LIN {X 0,Y 71.23,Z 524.249,A -85,B 0,C 180,E1 -30254.281,E2 -30254.281} C_VEL
LIN {X 0,Y 69.533,Z 525.783,A -85,B 0,C 180,E1 -30256.224,E2 -30256.224} C_VEL
LIN {X 0,Y 68.086,Z 526.954,A -85,B 0,C 180,E1 -30257.295,E2 -30257.295} C_VEL
LIN {X 0,Y 57.032,Z 533.486,A -85,B 0,C 180,E1 -30262.453,E2 -30262.453} C_VEL
LIN {X 0,Y 47.989,Z 537.812,A -85,B 0,C 180,E1 -30268.517,E2 -30268.517} C_VEL
LIN {X 0,Y 42.388,Z 540.184,A -85,B 0,C 180,E1 -30274.005,E2 -30274.005} C_VEL
LIN {X 0,Y 37.239,Z 541.987,A -85,B 0,C 180,E1 -30280.983,E2 -30280.983} C_VEL
LIN {X 0,Y 29.54,Z 544.455,A -85,B 0,C 180,E1 -30301.587,E2 -30301.587} C_VEL
LIN {X 0,Y 27.549,Z 545.056,A -85,B 0,C 180,E1 -30315.22,E2 -30315.22} C_VEL
LIN {X 0,Y 27.127,Z 545.222,A -85,B 0,C 180,E1 -30330,E2 -30330} C_VEL
LIN {X 0,Y 27.542,Z 545.056,A -85,B 0,C 180,E1 -30344.783,E2 -30344.783} C_VEL
LIN {X 0,Y 29.537,Z 544.455,A -85,B 0,C 180,E1 -30358.416,E2 -30358.416} C_VEL
LIN {X 0,Y 37.239,Z 541.987,A -85,B 0,C 180,E1 -30379.016,E2 -30379.016} C_VEL
LIN {X 0,Y 45.149,Z 539.032,A -85,B 0,C 180,E1 -30388.885,E2 -30388.885} C_VEL
LIN {X 0,Y 53.969,Z 535.041,A -85,B 0,C 180,E1 -30395.72,E2 -30395.72} C_VEL
LIN {X 0,Y 63.264,Z 529.907,A -85,B 0,C 180,E1 -30400.768,E2 -30400.768} C_VEL
LIN {X 0,Y 68.069,Z 526.953,A -85,B 0,C 180,E1 -30402.751,E2 -30402.751} C_VEL
LIN {X 0,Y 69.534,Z 525.783,A -85,B 0,C 180,E1 -30403.774,E2 -30403.774} C_VEL
LIN {X 0,Y 71.209,Z 524.264,A -85,B 0,C 180,E1 -30405.715,E2 -30405.715} C_VEL
LIN {X 0,Y 72.238,Z 522.956,A -85,B 0,C 180,E1 -30408.777,E2 -30408.777} C_VEL
LIN {X 0,Y 73.193,Z 521.436,A -85,B 0,C 180,E1 -30414.487,E2 -30414.487} C_VEL
LIN {X 0,Y 74.016,Z 520.373,A -85,B 0,C 180,E1 -30419.997,E2 -30419.997} C_VEL
LIN {X 0,Y 72.973,Z 521.245,A -85,B 0,C 180,E1 -30426.486,E2 -30426.486} C_VEL
LIN {X 0,Y 72.133,Z 522.493,A -85,B 0,C 180,E1 -30433.02,E2 -30433.02} C_VEL
LIN {X 0,Y 71.688,Z 523.511,A -85,B 0,C 180,E1 -30437.101,E2 -30437.101} C_VEL
LIN {X 0,Y 70.173,Z 526.051,A -85,B 0,C 180,E1 -30443.613,E2 -30443.613} C_VEL
LIN {X 0,Y 69.168,Z 527.484,A -85,B 0,C 180,E1 -30447.202,E2 -30447.202} C_VEL
LIN {X 0,Y 67.175,Z 530.211,A -85,B 0,C 180,E1 -30453.18,E2 -30453.18} C_VEL
LIN {X 0,Y 63.118,Z 534.913,A -85,B 0,C 180,E1 -30464.295,E2 -30464.295} C_VEL
LIN {X 0,Y 61.528,Z 538.124,A -85,B 0,C 180,E1 -30475.172,E2 -30475.172} C_VEL
LIN {X 0,Y 62.218,Z 540.119,A -85,B 0,C 180,E1 -30484.636,E2 -30484.636} C_VEL
LIN {X 0,Y 66.705,Z 541.924,A -85,B 0,C 180,E1 -30497.836,E2 -30497.836} C_VEL
LIN {X 0,Y 70.834,Z 542.361,A -85,B 0,C 180,E1 -30504.306,E2 -30504.306} C_VEL
LIN {X 0,Y 76.029,Z 542.359,A -85,B 0,C 180,E1 -30510,E2 -30510} C_VEL
LIN {X 0,Y 70.662,Z 542.338,A -85,B 0,C 180,E1 -30515.991,E2 -30515.991} C_VEL
LIN {X 0,Y 65.424,Z 541.656,A -85,B 0,C 180,E1 -30524.819,E2 -30524.819} C_VEL
LIN {X 0,Y 61.967,Z 539.777,A -85,B 0,C 180,E1 -30536.978,E2 -30536.978} C_VEL
LIN {X 0,Y 61.667,Z 537.523,A -85,B 0,C 180,E1 -30547.089,E2 -30547.089} C_VEL
LIN {X 0,Y 64.093,Z 533.66,A -85,B 0,C 180,E1 -30558.864,E2 -30558.864} C_VEL
LIN {X 0,Y 67.132,Z 530.214,A -85,B 0,C 180,E1 -30566.877,E2 -30566.877} C_VEL
LIN {X 0,Y 69.117,Z 527.515,A -85,B 0,C 180,E1 -30572.776,E2 -30572.776} C_VEL
LIN {X 0,Y 70.159,Z 526.06,A -85,B 0,C 180,E1 -30576.382,E2 -30576.382} C_VEL
LIN {X 0,Y 71.673,Z 523.521,A -85,B 0,C 180,E1 -30582.896,E2 -30582.896} C_VEL
LIN {X 0,Y 72.372,Z 522.086,A -85,B 0,C 180,E1 -30588.804,E2 -30588.804} C_VEL
LIN {X 0,Y 73.157,Z 521.071,A -85,B 0,C 180,E1 -30594.49,E2 -30594.49} C_VEL
LIN {X 0,Y 73.978,Z 520.403,A -85,B 0,C 180,E1 -30600.003,E2 -30600.003} C_VEL
LIN {X 0,Y 72.983,Z 521.692,A -85,B 0,C 180,E1 -30606.47,E2 -30606.47} C_VEL
LIN {X 0,Y 71.817,Z 522.781,A -85,B 0,C 180,E1 -30608.611,E2 -30608.611} C_VEL
LIN {X 0,Y 69.339,Z 524.72,A -85,B 0,C 180,E1 -30610.507,E2 -30610.507} C_VEL
LIN {X 0,Y 66.81,Z 526.482,A -85,B 0,C 180,E1 -30611.609,E2 -30611.609} C_VEL
LIN {X 0,Y 56.852,Z 532.194,A -85,B 0,C 180,E1 -30614.584,E2 -30614.584} C_VEL
LIN {X 0,Y 48.207,Z 536.373,A -85,B 0,C 180,E1 -30618.631,E2 -30618.631} C_VEL
LIN {X 0,Y 38.852,Z 539.986,A -85,B 0,C 180,E1 -30625.252,E2 -30625.252} C_VEL
LIN {X 0,Y 33.001,Z 541.789,A -85,B 0,C 180,E1 -30631.589,E2 -30631.589} C_VEL
LIN {X 0,Y 23.518,Z 544.257,A -85,B 0,C 180,E1 -30653.298,E2 -30653.298} C_VEL
LIN {X 0,Y 20.755,Z 544.859,A -85,B 0,C 180,E1 -30670.208,E2 -30670.208} C_VEL
LIN {X 0,Y 20.02,Z 545.025,A -85,B 0,C 180,E1 -30690,E2 -30690} C_VEL
LIN {X 0,Y 20.75,Z 544.859,A -85,B 0,C 180,E1 -30709.797,E2 -30709.797} C_VEL
LIN {X 0,Y 23.516,Z 544.257,A -85,B 0,C 180,E1 -30726.706,E2 -30726.706} C_VEL
LIN {X 0,Y 33.002,Z 541.789,A -85,B 0,C 180,E1 -30748.41,E2 -30748.41} C_VEL
LIN {X 0,Y 41.912,Z 538.834,A -85,B 0,C 180,E1 -30757.255,E2 -30757.255} C_VEL
LIN {X 0,Y 51.452,Z 534.843,A -85,B 0,C 180,E1 -30762.968,E2 -30762.968} C_VEL
LIN {X 0,Y 61.285,Z 529.709,A -85,B 0,C 180,E1 -30767.08,E2 -30767.08} C_VEL
LIN {X 0,Y 64.629,Z 527.791,A -85,B 0,C 180,E1 -30768.146,E2 -30768.146} C_VEL
LIN {X 0,Y 66.463,Z 526.233,A -85,B 0,C 180,E1 -30771.212,E2 -30771.212} C_VEL
LIN {X 0,Y 67.993,Z 524.44,A -85,B 0,C 180,E1 -30779.997,E2 -30779.997} C_VEL
LIN {X 0,Y 67.02,Z 525.123,A -85,B 0,C 180,E1 -30786.016,E2 -30786.016} C_VEL
LIN {X 0,Y 66.141,Z 526.239,A -85,B 0,C 180,E1 -30792.266,E2 -30792.266} C_VEL
LIN {X 0,Y 65.681,Z 526.931,A -85,B 0,C 180,E1 -30795.636,E2 -30795.636} C_VEL
LIN {X 0,Y 63.819,Z 529.051,A -85,B 0,C 180,E1 -30802.408,E2 -30802.408} C_VEL
LIN {X 0,Y 62.355,Z 530.751,A -85,B 0,C 180,E1 -30806.793,E2 -30806.793} C_VEL
LIN {X 0,Y 60.941,Z 532.143,A -85,B 0,C 180,E1 -30810.65,E2 -30810.65} C_VEL
LIN {X 0,Y 56.616,Z 536.128,A -85,B 0,C 180,E1 -30821.859,E2 -30821.859} C_VEL
LIN {X 0,Y 54.917,Z 538.355,A -85,B 0,C 180,E1 -30830.219,E2 -30830.219} C_VEL
LIN {X 0,Y 54.954,Z 540.749,A -85,B 0,C 180,E1 -30843.527,E2 -30843.527} C_VEL
LIN {X 0,Y 58.247,Z 542.165,A -85,B 0,C 180,E1 -30856.036,E2 -30856.036} C_VEL
LIN {X 0,Y 63.437,Z 542.703,A -85,B 0,C 180,E1 -30865.57,E2 -30865.57} C_VEL
LIN {X 0,Y 66.992,Z 542.61,A -85,B 0,C 180,E1 -30870,E2 -30870} C_VEL
LIN {X 0,Y 62.054,Z 542.606,A -85,B 0,C 180,E1 -30876.503,E2 -30876.503} C_VEL
LIN {X 0,Y 58.047,Z 542.141,A -85,B 0,C 180,E1 -30884.414,E2 -30884.414} C_VEL
LIN {X 0,Y 54.953,Z 540.75,A -85,B 0,C 180,E1 -30896.47,E2 -30896.47} C_VEL
LIN {X 0,Y 54.969,Z 538.321,A -85,B 0,C 180,E1 -30909.911,E2 -30909.911} C_VEL
LIN {X 0,Y 59.439,Z 533.499,A -85,B 0,C 180,E1 -30925.858,E2 -30925.858} C_VEL
LIN {X 0,Y 60.902,Z 532.155,A -85,B 0,C 180,E1 -30929.364,E2 -30929.364} C_VEL
LIN {X 0,Y 62.581,Z 530.469,A -85,B 0,C 180,E1 -30933.949,E2 -30933.949} C_VEL
LIN {X 0,Y 63.818,Z 529.043,A -85,B 0,C 180,E1 -30937.636,E2 -30937.636} C_VEL
LIN {X 0,Y 65.679,Z 526.932,A -85,B 0,C 180,E1 -30944.37,E2 -30944.37} C_VEL
LIN {X 0,Y 66.136,Z 526.243,A -85,B 0,C 180,E1 -30947.733,E2 -30947.733} C_VEL
LIN {X 0,Y 67.018,Z 525.125,A -85,B 0,C 180,E1 -30953.984,E2 -30953.984} C_VEL
LIN {X 0,Y 67.974,Z 524.453,A -85,B 0,C 180,E1 -30960.003,E2 -30960.003} C_VEL
LIN {X 0,Y 66.934,Z 525.57,A -85,B 0,C 180,E1 -30966.03,E2 -30966.03} C_VEL
LIN {X 0,Y 66.443,Z 526.249,A -85,B 0,C 180,E1 -30968.811,E2 -30968.811} C_VEL
LIN {X 0,Y 64.638,Z 527.792,A -85,B 0,C 180,E1 -30971.894,E2 -30971.894} C_VEL
LIN {X 0,Y 56.852,Z 532.194,A -85,B 0,C 180,E1 -30974.584,E2 -30974.584} C_VEL
LIN {X 0,Y 51.655,Z 534.66,A -85,B 0,C 180,E1 -30976.114,E2 -30976.114} C_VEL
LIN {X 0,Y 46.14,Z 536.86,A -85,B 0,C 180,E1 -30976.82,E2 -30976.82} C_VEL
LIN {X 0,Y 34.766,Z 540.354,A -85,B 0,C 180,E1 -30978.039,E2 -30978.039} C_VEL
LIN {X 0,Y 28.325,Z 542.039,A -85,B 0,C 180,E1 -30981.502,E2 -30981.502} C_VEL
LIN {X 0,Y 27.465,Z 542.133,A -85,B 0,C 180,E1 -30982.411,E2 -30982.411} C_VEL
LIN {X 0,Y 18.313,Z 544.06,A -85,B 0,C 180,E1 -30999.867,E2 -30999.867} C_VEL
LIN {X 0,Y 14.258,Z 544.661,A -85,B 0,C 180,E1 -31020.468,E2 -31020.468} C_VEL
LIN {X 0,Y 12.927,Z 544.828,A -85,B 0,C 180,E1 -31050,E2 -31050} C_VEL
LIN {X 0,Y 14.254,Z 544.661,A -85,B 0,C 180,E1 -31079.54,E2 -31079.54} C_VEL
LIN {X 0,Y 18.311,Z 544.059,A -85,B 0,C 180,E1 -31100.138,E2 -31100.138} C_VEL
LIN {X 0,Y 29.89,Z 541.591,A -85,B 0,C 180,E1 -31120.134,E2 -31120.134} C_VEL
LIN {X 0,Y 39.705,Z 538.636,A -85,B 0,C 180,E1 -31126.782,E2 -31126.782} C_VEL
LIN {X 0,Y 49.829,Z 534.645,A -85,B 0,C 180,E1 -31130.849,E2 -31130.849} C_VEL
LIN {X 0,Y 58.983,Z 530.129,A -85,B 0,C 180,E1 -31133.466,E2 -31133.466} C_VEL
LIN {X 0,Y 60.842,Z 528.987,A -85,B 0,C 180,E1 -31135.177,E2 -31135.177} C_VEL
LIN {X 0,Y 61.729,Z 528.247,A -85,B 0,C 180,E1 -31139.996,E2 -31139.996} C_VEL
LIN {X 0,Y 60.611,Z 528.88,A -85,B 0,C 180,E1 -31146.655,E2 -31146.655} C_VEL
LIN {X 0,Y 59.556,Z 529.947,A -85,B 0,C 180,E1 -31153.648,E2 -31153.648} C_VEL
LIN {X 0,Y 58.739,Z 530.76,A -85,B 0,C 180,E1 -31156.83,E2 -31156.83} C_VEL
LIN {X 0,Y 57.078,Z 532.15,A -85,B 0,C 180,E1 -31161.674,E2 -31161.674} C_VEL
LIN {X 0,Y 55.102,Z 533.736,A -85,B 0,C 180,E1 -31166.774,E2 -31166.774} C_VEL
LIN {X 0,Y 51.518,Z 536.355,A -85,B 0,C 180,E1 -31175.066,E2 -31175.066} C_VEL
LIN {X 0,Y 48.361,Z 539.037,A -85,B 0,C 180,E1 -31186.597,E2 -31186.597} C_VEL
LIN {X 0,Y 47.898,Z 541.491,A -85,B 0,C 180,E1 -31203.885,E2 -31203.885} C_VEL
LIN {X 0,Y 50.672,Z 542.526,A -85,B 0,C 180,E1 -31216.12,E2 -31216.12} C_VEL
LIN {X 0,Y 58.08,Z 542.857,A -85,B 0,C 180,E1 -31230,E2 -31230} C_VEL
LIN {X 0,Y 50.67,Z 542.527,A -85,B 0,C 180,E1 -31243.874,E2 -31243.874} C_VEL
LIN {X 0,Y 47.729,Z 541.3,A -85,B 0,C 180,E1 -31257.944,E2 -31257.944} C_VEL
LIN {X 0,Y 48.89,Z 538.582,A -85,B 0,C 180,E1 -31275.95,E2 -31275.95} C_VEL
LIN {X 0,Y 52.745,Z 535.549,A -85,B 0,C 180,E1 -31287.798,E2 -31287.798} C_VEL
LIN {X 0,Y 55.083,Z 533.737,A -85,B 0,C 180,E1 -31293.265,E2 -31293.265} C_VEL
LIN {X 0,Y 57.043,Z 532.166,A -85,B 0,C 180,E1 -31298.312,E2 -31298.312} C_VEL
LIN {X 0,Y 58.722,Z 530.761,A -85,B 0,C 180,E1 -31303.223,E2 -31303.223} C_VEL
LIN {X 0,Y 59.552,Z 529.949,A -85,B 0,C 180,E1 -31306.352,E2 -31306.352} C_VEL
LIN {X 0,Y 60.609,Z 528.881,A -85,B 0,C 180,E1 -31313.345,E2 -31313.345} C_VEL
LIN {X 0,Y 61.714,Z 528.256,A -85,B 0,C 180,E1 -31320.004,E2 -31320.004} C_VEL
LIN {X 0,Y 60.842,Z 528.986,A -85,B 0,C 180,E1 -31324.819,E2 -31324.819} C_VEL
LIN {X 0,Y 58.984,Z 530.13,A -85,B 0,C 180,E1 -31326.542,E2 -31326.542} C_VEL
LIN {X 0,Y 49.829,Z 534.645,A -85,B 0,C 180,E1 -31329.15,E2 -31329.15} C_VEL
LIN {X 0,Y 39.703,Z 538.636,A -85,B 0,C 180,E1 -31333.205,E2 -31333.205} C_VEL
LIN {X 0,Y 29.89,Z 541.591,A -85,B 0,C 180,E1 -31339.863,E2 -31339.863} C_VEL
LIN {X 0,Y 27.465,Z 542.133,A -85,B 0,C 180,E1 -31342.411,E2 -31342.411} C_VEL
LIN {X 0,Y 22.212,Z 543.248,A -85,B 0,C 180,E1 -31348.217,E2 -31348.217} C_VEL
LIN {X 0,Y 16.762,Z 544.025,A -85,B 0,C 180,E1 -31354.874,E2 -31354.874} C_VEL
LIN {X 0,Y 7.018,Z 544.655,A -85,B 0,C 180,E1 -31392.355,E2 -31392.355} C_VEL
LIN {X 0,Y 7.891,Z 544.494,A -85,B 0,C 180,E1 -31456.951,E2 -31456.951} C_VEL
LIN {X 0,Y 14.792,Z 543.862,A -85,B 0,C 180,E1 -31481.847,E2 -31481.847} C_VEL
LIN {X 0,Y 28.274,Z 541.394,A -85,B 0,C 180,E1 -31493.842,E2 -31493.842} C_VEL
LIN {X 0,Y 38.702,Z 538.438,A -85,B 0,C 180,E1 -31497.128,E2 -31497.128} C_VEL
LIN {X 0,Y 49.201,Z 534.447,A -85,B 0,C 180,E1 -31499.082,E2 -31499.082} C_VEL
LIN {X 0,Y 55.271,Z 531.728,A -85,B 0,C 180,E1 -31499.996,E2 -31499.996} C_VEL
LIN {X 0,Y 53.96,Z 532.338,A -85,B 0,C 180,E1 -31507.479,E2 -31507.479} C_VEL
LIN {X 0,Y 51.998,Z 533.654,A -85,B 0,C 180,E1 -31515.679,E2 -31515.679} C_VEL
LIN {X 0,Y 49.39,Z 535.425,A -85,B 0,C 180,E1 -31522.357,E2 -31522.357} C_VEL
LIN {X 0,Y 43.573,Z 538.811,A -85,B 0,C 180,E1 -31536.25,E2 -31536.25} C_VEL
LIN {X 0,Y 41.18,Z 540.475,A -85,B 0,C 180,E1 -31546.95,E2 -31546.95} C_VEL
LIN {X 0,Y 41.749,Z 542.643,A -85,B 0,C 180,E1 -31570.326,E2 -31570.326} C_VEL
LIN {X 0,Y 44.714,Z 543.091,A -85,B 0,C 180,E1 -31580.957,E2 -31580.957} C_VEL
LIN {X 0,Y 49.192,Z 543.104,A -85,B 0,C 180,E1 -31590.093,E2 -31590.093} C_VEL
LIN {X 0,Y 43.306,Z 542.91,A -85,B 0,C 180,E1 -31603.187,E2 -31603.187} C_VEL
LIN {X 0,Y 40.547,Z 541.724,A -85,B 0,C 180,E1 -31621.33,E2 -31621.33} C_VEL
LIN {X 0,Y 42.078,Z 539.718,A -85,B 0,C 180,E1 -31638.088,E2 -31638.088} C_VEL
LIN {X 0,Y 47.495,Z 536.456,A -85,B 0,C 180,E1 -31653.651,E2 -31653.651} C_VEL
LIN {X 0,Y 49.379,Z 535.426,A -85,B 0,C 180,E1 -31657.675,E2 -31657.675} C_VEL
LIN {X 0,Y 51.955,Z 533.673,A -85,B 0,C 180,E1 -31664.308,E2 -31664.308} C_VEL
LIN {X 0,Y 53.959,Z 532.339,A -85,B 0,C 180,E1 -31672.52,E2 -31672.52} C_VEL
LIN {X 0,Y 55.11,Z 531.807,A -85,B 0,C 180,E1 -31680.004,E2 -31680.004} C_VEL
LIN {X 0,Y 45.696,Z 535.978,A -85,B 0,C 180,E1 -31681.468,E2 -31681.468} C_VEL
LIN {X 0,Y 35.216,Z 539.59,A -85,B 0,C 180,E1 -31683.789,E2 -31683.789} C_VEL
LIN {X 0,Y 24.827,Z 542.094,A -85,B 0,C 180,E1 -31687.937,E2 -31687.937} C_VEL
LIN {X 0,Y 14.792,Z 543.862,A -85,B 0,C 180,E1 -31698.159,E2 -31698.159} C_VEL
LIN {X 0,Y 8.799,Z 544.464,A -85,B 0,C 180,E1 -31716.995,E2 -31716.995} C_VEL
LIN {X 0,Y 5.821,Z 544.631,A -85,B 0,C 180,E1 -31770,E2 -31770} C_VEL
LIN {X 0,Y 7.891,Z 544.494,A -85,B 0,C 180,E1 -31816.951,E2 -31816.951} C_VEL
LIN {X 0,Y 12.278,Z 544.146,A -85,B 0,C 180,E1 -31839.888,E2 -31839.888} C_VEL
LIN {X 0,Y 20.568,Z 542.828,A -85,B 0,C 180,E1 -31858.93,E2 -31858.93} C_VEL
LIN {X 0,Y 29.705,Z 540.885,A -85,B 0,C 180,E1 -31866.809,E2 -31866.809} C_VEL
LIN {X 0,Y 35.428,Z 539.402,A -85,B 0,C 180,E1 -31867.76,E2 -31867.76} C_VEL
LIN {X 0,Y 42.538,Z 537.021,A -85,B 0,C 180,E1 -31867.569,E2 -31867.569} C_VEL
LIN {X 0,Y 46.706,Z 535.551,A -85,B 0,C 180,E1 -31868.65,E2 -31868.65} C_VEL
LIN {X 0,Y 44.011,Z 536.827,A -85,B 0,C 180,E1 -31876.646,E2 -31876.646} C_VEL
LIN {X 0,Y 39.292,Z 539.038,A -85,B 0,C 180,E1 -31886.581,E2 -31886.581} C_VEL
LIN {X 0,Y 35.596,Z 540.704,A -85,B 0,C 180,E1 -31897.84,E2 -31897.84} C_VEL
LIN {X 0,Y 33.848,Z 542.879,A -85,B 0,C 180,E1 -31925.464,E2 -31925.464} C_VEL
LIN {X 0,Y 36.229,Z 543.331,A -85,B 0,C 180,E1 -31938.815,E2 -31938.815} C_VEL
LIN {X 0,Y 40.519,Z 543.345,A -85,B 0,C 180,E1 -31950,E2 -31950} C_VEL
LIN {X 0,Y 35.951,Z 543.293,A -85,B 0,C 180,E1 -31962.224,E2 -31962.224} C_VEL
LIN {X 0,Y 33.511,Z 542.379,A -85,B 0,C 180,E1 -31982.989,E2 -31982.989} C_VEL
LIN {X 0,Y 36.188,Z 540.394,A -85,B 0,C 180,E1 -32004.372,E2 -32004.372} C_VEL
LIN {X 0,Y 39.307,Z 539.037,A -85,B 0,C 180,E1 -32013.376,E2 -32013.376} C_VEL
LIN {X 0,Y 44.002,Z 536.827,A -85,B 0,C 180,E1 -32023.395,E2 -32023.395} C_VEL
LIN {X 0,Y 46.689,Z 535.558,A -85,B 0,C 180,E1 -32031.347,E2 -32031.347} C_VEL
LIN {X 0,Y 42.539,Z 537.021,A -85,B 0,C 180,E1 -32032.417,E2 -32032.417} C_VEL
LIN {X 0,Y 35.465,Z 539.393,A -85,B 0,C 180,E1 -32032.232,E2 -32032.232} C_VEL
LIN {X 0,Y 28.407,Z 541.196,A -85,B 0,C 180,E1 -32031.727,E2 -32031.727} C_VEL
LIN {X 0,Y 14.282,Z 543.663,A -85,B 0,C 180,E1 -32029.785,E2 -32029.785} C_VEL
LIN {X 0,Y 7.264,Z 544.266,A -85,B 0,C 180,E1 -32025.355,E2 -32025.355} C_VEL
LIN {X 0,Y 1.291,Z 544.433,A -85,B 0,C 180,E1 -31950,E2 -31950} C_VEL
LIN {X 0,Y 7.265,Z 544.266,A -85,B 0,C 180,E1 -31874.671,E2 -31874.671} C_VEL
LIN {X 0,Y 14.282,Z 543.663,A -85,B 0,C 180,E1 -31870.221,E2 -31870.221} C_VEL
LIN {X 0,Y 28.407,Z 541.196,A -85,B 0,C 180,E1 -31868.269,E2 -31868.269} C_VEL
LIN {X 0,Y 35.428,Z 539.402,A -85,B 0,C 180,E1 -31867.76,E2 -31867.76} C_VEL
LIN {X 0,Y 34.515,Z 539.694,A -85,B 0,C 180,E1 -31869.653,E2 -31869.653} C_VEL
LIN {X 0,Y 28.379,Z 541.288,A -85,B 0,C 180,E1 -31875.235,E2 -31875.235} C_VEL
LIN {X 0,Y 18.092,Z 543.305,A -85,B 0,C 180,E1 -31888.713,E2 -31888.713} C_VEL
LIN {X 0,Y 11.41,Z 544.061,A -85,B 0,C 180,E1 -31911.263,E2 -31911.263} C_VEL
LIN {X 0,Y 9.703,Z 544.135,A -85,B 0,C 180,E1 -31924.188,E2 -31924.188} C_VEL
LIN {X 0,Y 8.391,Z 544.236,A -85,B 0,C 180,E1 -31950,E2 -31950} C_VEL
LIN {X 0,Y 11.387,Z 544.068,A -85,B 0,C 180,E1 -31988.109,E2 -31988.109} C_VEL
LIN {X 0,Y 17.061,Z 543.465,A -85,B 0,C 180,E1 -32005.472,E2 -32005.472} C_VEL
LIN {X 0,Y 30.261,Z 540.999,A -85,B 0,C 180,E1 -32018.275,E2 -32018.275} C_VEL
LIN {X 0,Y 32.626,Z 540.445,A -85,B 0,C 180,E1 -32017.587,E2 -32017.587} C_VEL
LIN {X 0,Y 26.58,Z 542.914,A -85,B 0,C 180,E1 -31987.526,E2 -31987.526} C_VEL
LIN {X 0,Y 28.621,Z 543.658,A -85,B 0,C 180,E1 -31960.863,E2 -31960.863} C_VEL
LIN {X 0,Y 31.831,Z 543.586,A -85,B 0,C 180,E1 -31950,E2 -31950} C_VEL
LIN {X 0,Y 27.905,Z 543.567,A -85,B 0,C 180,E1 -31935.413,E2 -31935.413} C_VEL
LIN {X 0,Y 26.522,Z 542.929,A -85,B 0,C 180,E1 -31912.639,E2 -31912.639} C_VEL
LIN {X 0,Y 32.594,Z 540.453,A -85,B 0,C 180,E1 -31882.422,E2 -31882.422} C_VEL
LIN {X 0,Y 30.26,Z 540.999,A -85,B 0,C 180,E1 -31881.721,E2 -31881.721} C_VEL
LIN {X 0,Y 17.062,Z 543.465,A -85,B 0,C 180,E1 -31894.531,E2 -31894.531} C_VEL
LIN {X 0,Y 9.703,Z 544.135,A -85,B 0,C 180,E1 -31924.188,E2 -31924.188} C_VEL
LIN {X 0,Y 9.118,Z 544.22,A -85,B 0,C 180,E1 -31948.452,E2 -31948.452} C_VEL
LIN {X 0,Y 11.105,Z 544.177,A -85,B 0,C 180,E1 -31968.666,E2 -31968.666} C_VEL
LIN {X 0,Y 15.017,Z 543.954,A -85,B 0,C 180,E1 -31980.065,E2 -31980.065} C_VEL
LIN {X 0,Y 17.776,Z 543.741,A -85,B 0,C 180,E1 -31980.979,E2 -31980.979} C_VEL
LIN {X 0,Y 19.28,Z 543.666,A -85,B 0,C 180,E1 -31978.672,E2 -31978.672} C_VEL
LIN {X 0,Y 19.493,Z 543.678,A -85,B 0,C 180,E1 -31977.286,E2 -31977.286} C_VEL
LIN {X 0,Y 23.221,Z 543.825,A -85,B 0,C 180,E1 -31950,E2 -31950} C_VEL
LIN {X 0,Y 19.46,Z 543.682,A -85,B 0,C 180,E1 -31922.813,E2 -31922.813} C_VEL
LIN {X 0,Y 17.546,Z 543.871,A -85,B 0,C 180,E1 -31926.388,E2 -31926.388} C_VEL
LIN {X 0,Y 15.509,Z 544.039,A -85,B 0,C 180,E1 -31950,E2 -31950} C_VEL
LIN {X 0,Y 17.544,Z 543.871,A -85,B 0,C 180,E1 -31973.615,E2 -31973.615} C_VEL
LIN {X 0,Y 19.493,Z 543.678,A -85,B 0,C 180,E1 -31977.286,E2 -31977.286} C_VEL
LIN {X 0,Y 21.408,Z 545.671,A -85,B 0,C 180,E1 -31980.144,E2 -31980.144} C_VEL
LIN {X 0,Y 21.408,Z 600,A -85,B 0,C 180,E1 -31980.144,E2 -31980.144} C_VEL
LIN {X 0,Y 21.408,Z 600,A -85,B 0,C 180,E1 -31980.144,E2 -31980.144}

QRS_NEXT_CUT()

QRS_NEXT()
QRS_HOME()

END
